(* CoDeSys 2.3.9.45 project: Stromsensor_01.pro *)
(* Libraries: SerComm.lib*31.5.11 08:54:36, Serial_Interface_01.lib*22.4.13 12:50:14, Modb_l05.lib*22.4.13 12:50:12, mod_com.lib*2.12.10 14:48:32, Standard.lib 20.5.14 08:13:26, Iecsfc.lib 16.5.13 14:00:50, SYSLIBCALLBACK.LIB 16.5.13 14:00:50 *)

(* Global variable list: Global_Constant *)
VAR_GLOBAL CONSTANT

	(*--- this values are possible parameters -> the real used quantity of sensors have to be smaller or equal ---*)
	MAX_SENSORS_PER_LINE		:	BYTE := 32;	(* max. quantity of possible slaves per line *)
	(*----------------------------------------------------------------------------------------------------------------------------------------------------------*)

END_VAR

(* Data type in line information/current sensor *)
TYPE typCurrentSensor :
	STRUCT
		rActualCurrent				:	REAL 	:= 0.0;	(* [A] actual  current *)
		rLimitErrorCurrent			:	REAL 	:= -3.0;	(* [A] threshold parameter for negative current error *)
		rInstalledCurrent			:	REAL 	:= 0.0; 	(* [A] installed nominal 125% current *)
		udErrorCounter			:	UDINT	:= 0;	(* error counter *)
		bErrorMaster				:	BYTE	:= 0;	(* communication error -> detected by the master *)
		bErrorSlave				:	BYTE	:= 0;	(* error at this sensor ->error generated and reprted by this slave *)

		bFillByte					:	BYTE 	:= 0;	(* fill byte to have an even byte count for this structure *)

		bSlaveAddress			:	BYTE	:= 0;	(* modbus address of this slave *)

		rBargraphValue			:	REAL 	:= 0.0;	(* value for Bargraph range -3.0 .. 80.0 *)


		xErrorMaster				:	BOOL;			(* error at this sensor -> see bErrorMaster *)
		xErrorSlave				:	BOOL;			(* error at this sensor -> see cErrorSlave *)
		xErrorOverflow				:	BOOL;			(* error at this sensor -> see 125% value *)
		xErrorUnderflow			:	BOOL;			(* error at this sensor -> see min. limit value *)
		xResetErrorCounter		:	BOOL;

		sDescription				:	STRING(25);	(* free userdefined description for this sensor *)
	END_STRUCT
END_TYPE

(* Data type in line information *)
TYPE typLineInfo :
	STRUCT
		Sensors 	:	ARRAY[1..MAX_SENSORS_PER_LINE] OF typCurrentSensor :=
									(*--- init values ------------------------------------------------------------------------------*)
									(rLimitErrorCurrent := -3.0, rInstalledCurrent := 29.8, bSlaveAddress := 1),
									(rLimitErrorCurrent := -3.0, rInstalledCurrent := 29.8, bSlaveAddress := 2),
									(rLimitErrorCurrent := -3.0, rInstalledCurrent := 29.8, bSlaveAddress := 3),
									(rLimitErrorCurrent := -3.0, rInstalledCurrent := 29.8, bSlaveAddress := 4),
									(rLimitErrorCurrent := -3.0, rInstalledCurrent := 29.8, bSlaveAddress := 5),
									(rLimitErrorCurrent := -3.0, rInstalledCurrent := 29.8, bSlaveAddress := 6),
									(rLimitErrorCurrent := -3.0, rInstalledCurrent := 29.8, bSlaveAddress := 7),
									(rLimitErrorCurrent := -3.0, rInstalledCurrent := 29.8, bSlaveAddress := 8),
									(rLimitErrorCurrent := -3.0, rInstalledCurrent := 29.8, bSlaveAddress := 9),
									(rLimitErrorCurrent := -3.0, rInstalledCurrent := 29.8, bSlaveAddress := 10),
									(rLimitErrorCurrent := -3.0, rInstalledCurrent := 29.8, bSlaveAddress := 11),
									(rLimitErrorCurrent := -3.0, rInstalledCurrent := 29.8, bSlaveAddress := 12),
									(rLimitErrorCurrent := -3.0, rInstalledCurrent := 29.8, bSlaveAddress := 13),
									(rLimitErrorCurrent := -3.0, rInstalledCurrent := 29.8, bSlaveAddress := 14),
									(rLimitErrorCurrent := -3.0, rInstalledCurrent := 29.8, bSlaveAddress := 15),
									(rLimitErrorCurrent := -3.0, rInstalledCurrent := 29.8, bSlaveAddress := 16),
									(rLimitErrorCurrent := -3.0, rInstalledCurrent := 29.8, bSlaveAddress := 17),
									(rLimitErrorCurrent := -3.0, rInstalledCurrent := 29.8, bSlaveAddress := 18),
									(rLimitErrorCurrent := -3.0, rInstalledCurrent := 29.8, bSlaveAddress := 19),
									(rLimitErrorCurrent := -3.0, rInstalledCurrent := 29.8, bSlaveAddress := 20),
									(rLimitErrorCurrent := -3.0, rInstalledCurrent := 29.8, bSlaveAddress := 21),
									(rLimitErrorCurrent := -3.0, rInstalledCurrent := 29.8, bSlaveAddress := 22),
									(rLimitErrorCurrent := -3.0, rInstalledCurrent := 29.8, bSlaveAddress := 23),
									(rLimitErrorCurrent := -3.0, rInstalledCurrent := 29.8, bSlaveAddress := 24),
									(rLimitErrorCurrent := -3.0, rInstalledCurrent := 29.8, bSlaveAddress := 25),
									(rLimitErrorCurrent := -3.0, rInstalledCurrent := 29.8, bSlaveAddress := 26),
									(rLimitErrorCurrent := -3.0, rInstalledCurrent := 29.8, bSlaveAddress := 27),
									(rLimitErrorCurrent := -3.0, rInstalledCurrent := 29.8, bSlaveAddress := 28),
									(rLimitErrorCurrent := -3.0, rInstalledCurrent := 29.8, bSlaveAddress := 29),
									(rLimitErrorCurrent := -3.0, rInstalledCurrent := 29.8, bSlaveAddress := 30),
									(rLimitErrorCurrent := -3.0, rInstalledCurrent := 29.8, bSlaveAddress := 31),
									(rLimitErrorCurrent := -3.0, rInstalledCurrent := 29.8, bSlaveAddress := 32);
									(*--------------------------------------------------------------------------------------------------*)
	END_STRUCT
END_TYPE

(* POU PLC_PRG, FBD *)
PROGRAM PLC_PRG
VAR RETAIN PERSISTENT
	SensorQuantity		:	BYTE := 1;			(* quantity of sensors -> 1 .. 32 *)
	Line					:	typLineInfo; 		(* table data *)
END_VAR
VAR
	mySensorLine		:	MODBUS_LINE;   (* communication fb *)
END_VAR
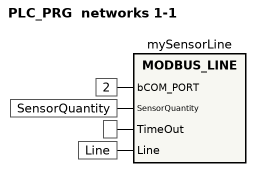
_FBD_ (* Function Block Diagram *)
NETWORK 1
	mySensorLine:MODBUS_LINE(bCOM_PORT: 2, SensorQuantity: SensorQuantity, TimeOut: , Line: Line)
_END_FBD_
END_PROGRAM

(* POU Line Communication/Single Line/MODBUS_LINE, ST *)
FUNCTION_BLOCK MODBUS_LINE
(*--- INTERFACE VARIABLES -------------------------------------------------------------------------------------*)
VAR_INPUT
	bCOM_PORT		:	BYTE := 2;
	SensorQuantity	:	BYTE := 1;			(* quantity of sensors *)
	TimeOut			:	TIME := t#30ms;	(* timeout for communication *)
END_VAR
VAR_IN_OUT
	Line				:	typLineInfo;		(**)
END_VAR
(*--- END INTERFACE VARIABLES ------------------------------------------------------------------------------*)

(*--- LOCAL VARIABLES --------------------------------------------------------------------------------------------*)
VAR
	MB_Master		:	MODBUS_MASTER_RTU;
	Query				:	typModbusQuery := (SlaveAddress := 1, FunctionCode := 3, StartAddress := 4, Quantity := 1, Data := 125(0) ); (* default values *)
	Start				:	BOOL;
	Response			:	typModbusResponse;

	JobNr				:	INT := 0;
	JobDelay			:	TON := (PT := t#30ms);
	i					:	INT;
	JobActive			:	BOOL;
END_VAR
(*--- delay between  two requests -----------------------*)
JobDelay(IN := NOT Start ); (*, PT := t#30ms);*)
(*-------------------------------------------------------------------*)

(*--- start a request  ------------------------------------------------------------------------------------*)
IF JobDelay.Q OR ((MB_Master.MB_Error = MB_TIME_OUT) AND NOT Start) THEN (* next job  *)
	JobNr := (JobNr MOD SensorQuantity) + 1;
	Query.SlaveAddress := Line.Sensors[JobNr].bSlaveAddress;

	Start := (Query.SlaveAddress <> 0);  (* if address <> 0 then start a request *)
	JobActive := Start;
END_IF
(*----------------------------------------------------------------------------------------------------------------------------*)

(*--- call the modbus master  ----------------------------------------------*)
MB_Master(	bCOM_PORT					:= bCOM_PORT,
				cbCOM_BAUDRATE			:= BAUD_19200,
				cpCOM_PARITY				:= PARITY_EVEN,
				csCOM_STOPBITS			:= STOPBITS_1,
				cbsCOM_BYTESIZE			:= BS_8,
				cfCOM_FLOW_CONTROL	:= HALFDUPLEX,
				TimeOut						:= TimeOut,
				StartFunction					:= Start,
				Query							:= Query,
				Response						:= Response);
(*------------------------------------------------------------------------------------*)

(*--- take over the response from sensor ----------------------------------------------------------------------------------------------*)
IF NOT Start AND (JobNr >= 1) AND (JobNr <= MAX_SENSORS_PER_LINE) AND JobActive THEN (* job is ready *)
	JobActive := FALSE;

	(*--- special process for  address 0 ------------------------------------------------------------*)
	IF Line.Sensors[JobNr].bSlaveAddress = 0  THEN (* Address = 0 -> erase errors *)
		Line.Sensors[JobNr].bErrorMaster 		:= 0;
		Line.Sensors[JobNr].bErrorSlave 		:= 0;
		Line.Sensors[JobNr].rActualCurrent 		:= 0.0; (* delete value  *)
		Line.Sensors[JobNr].rBargraphValue 	:= 0.0; (* delete bargraph *)
	(*----------------------------------------------------------------------------------------------------------*)

	ELSE (* take over the data  *)
		Line.Sensors[JobNr].bErrorMaster := INT_TO_BYTE(MB_Master.MB_Error);
		Line.Sensors[JobNr].bErrorSlave := WORD_TO_BYTE(Response.Error);

		IF MB_Master.MB_Error = MB_NO_ERROR THEN (* Job OK -> no errors -> take over the value  *)
			Line.Sensors[JobNr].rActualCurrent := INC_TO_AMPERE(Response.Data[0]); (* convert increments to ampere *)
			(*--- scale bargraph for 125%  -------------------------------------------------------------------------------------------------------------*)
			IF (Line.Sensors[JobNr].rInstalledCurrent > 0)  (* NO DIV 0 !!!  *)
			AND (Line.Sensors[JobNr].rActualCurrent > 0) THEN

				Line.Sensors[JobNr].rBargraphValue := (80.0 / Line.Sensors[JobNr].rInstalledCurrent) * Line.Sensors[JobNr].rActualCurrent;
			ELSE (* !! DIV durch NULL *)
				Line.Sensors[JobNr].rBargraphValue := Line.Sensors[JobNr].rActualCurrent;
			END_IF
			(*----------------------------------------------------------------------------------------------------------------------------------------------------*)

		ELSE (* error -> delete values *)
			Line.Sensors[JobNr].rActualCurrent 		:= 0.0;
			Line.Sensors[JobNr].rBargraphValue 	:= 0.0;

		END_IF
	END_IF

	ERROR_COUNTER; (* increment errorcounter  *)

END_IF

(*--- reset error counter ----------------------------------*)
FOR i := 1 TO SensorQuantity DO
	IF Line.Sensors[i].xResetErrorCounter THEN
		Line.Sensors[i].xResetErrorCounter := FALSE;
		Line.Sensors[i].udErrorCounter := 0;
	END_IF
END_FOR
(*---------------------------------------------------------------*)
END_FUNCTION_BLOCK
ACTION ERROR_COUNTER:
(*--- check for errors  --------------------------------------------------------------------------------------------------------------------------------------*)
Line.Sensors[JobNr].xErrorMaster 		:= (Line.Sensors[JobNr].bErrorMaster <> 0);
Line.Sensors[JobNr].xErrorSlave 		:= (Line.Sensors[JobNr].bErrorSlave <> 0);
Line.Sensors[JobNr].xErrorOverflow 		:= (Line.Sensors[JobNr].rActualCurrent > Line.Sensors[JobNr].rInstalledCurrent);
Line.Sensors[JobNr].xErrorUnderflow 	:= (Line.Sensors[JobNr].rActualCurrent < Line.Sensors[JobNr].rLimitErrorCurrent);

IF 	Line.Sensors[JobNr].xErrorMaster
	OR Line.Sensors[JobNr].xErrorSlave
	OR Line.Sensors[JobNr].xErrorOverflow
	OR Line.Sensors[JobNr].xErrorUnderflow
	 THEN (* increment error counter *)
	Line.Sensors[JobNr].udErrorCounter := Line.Sensors[JobNr].udErrorCounter + 1;
END_IF
END_ACTION

(* POU Line Communication/Single Line/Helper/INC_TO_AMPERE, ST *)
FUNCTION INC_TO_AMPERE : REAL
VAR_INPUT
	IN		:	WORD;
END_VAR
(* calculation from increments to ampere *)
INC_TO_AMPERE := (80.0 		(* max. current *)
                                       / 29126)	(* -> 32767 - 3641  Increments of the module for MAX_CURRENT *)
						* WORD_TO_INT(IN);
END_FUNCTION

(* Visualisation MASTER FOLIE/MASTERFOLIE
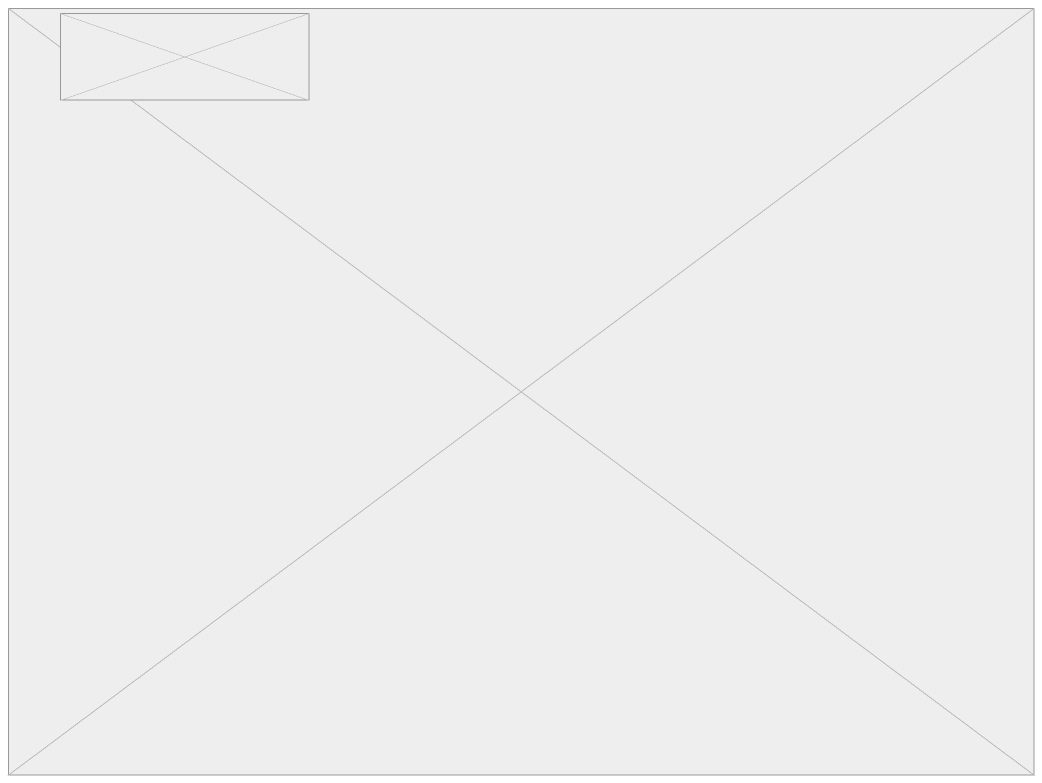
bitmap at (-1,0)-(1025,767): BILDER\789_620.BMP
bitmap at (51,5)-(300,92): BILDER\WAGO_INO.BMP
*)

(* Visualisation PLC_VISU
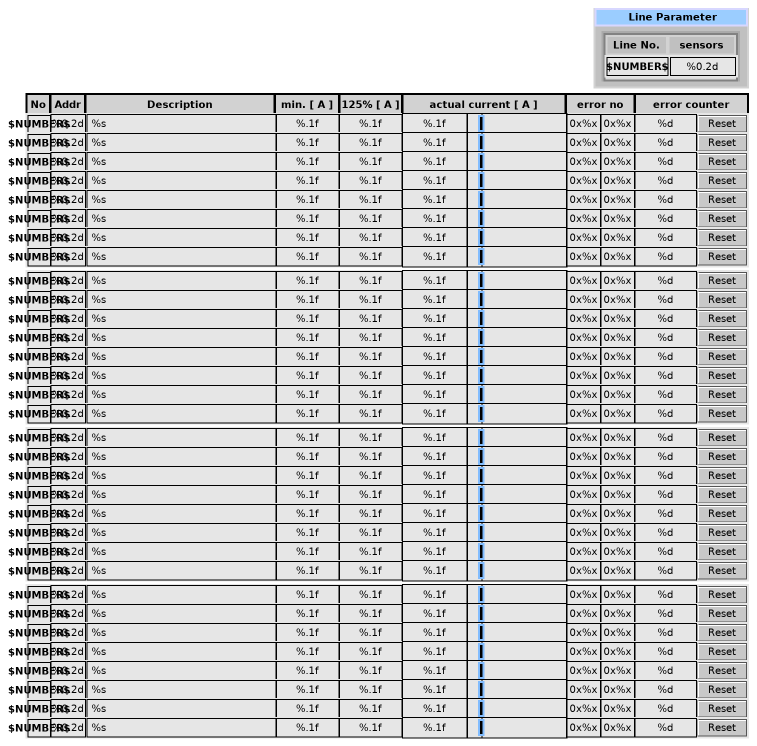
embedded screen at (51,92)-(774,116): VISU_TABLE_HEADLINE
embedded screen at (51,113)-(774,134): VISU_LINE
embedded screen at (51,132)-(774,153): VISU_LINE
embedded screen at (51,151)-(774,172): VISU_LINE
embedded screen at (51,170)-(774,191): VISU_LINE
embedded screen at (51,189)-(774,210): VISU_LINE
embedded screen at (51,208)-(774,229): VISU_LINE
embedded screen at (51,227)-(774,248): VISU_LINE
embedded screen at (51,246)-(774,267): VISU_LINE
embedded screen at (51,270)-(774,291): VISU_LINE
embedded screen at (51,289)-(774,310): VISU_LINE
embedded screen at (51,308)-(774,329): VISU_LINE
embedded screen at (51,327)-(774,348): VISU_LINE
embedded screen at (51,346)-(774,367): VISU_LINE
embedded screen at (51,365)-(774,386): VISU_LINE
embedded screen at (51,384)-(774,405): VISU_LINE
embedded screen at (51,403)-(774,424): VISU_LINE
embedded screen at (51,427)-(774,448): VISU_LINE
embedded screen at (51,446)-(774,467): VISU_LINE
embedded screen at (51,465)-(774,486): VISU_LINE
embedded screen at (51,484)-(774,505): VISU_LINE
embedded screen at (51,503)-(774,524): VISU_LINE
embedded screen at (51,522)-(774,543): VISU_LINE
embedded screen at (51,541)-(774,562): VISU_LINE
embedded screen at (51,560)-(774,581): VISU_LINE
embedded screen at (51,584)-(774,605): VISU_LINE
embedded screen at (51,603)-(774,624): VISU_LINE
embedded screen at (51,622)-(774,643): VISU_LINE
embedded screen at (51,641)-(774,662): VISU_LINE
embedded screen at (51,660)-(774,681): VISU_LINE
embedded screen at (51,679)-(774,700): VISU_LINE
embedded screen at (51,698)-(774,719): VISU_LINE
embedded screen at (51,717)-(774,738): VISU_LINE
group at (619,8)-(774,88)
  rectangle at (1,0)-(154,18): text "Line Parameter"
  rectangle at (12,27)-(74,47): text "Line No."
  rectangle at (74,27)-(142,47): text "sensors"
  embedded screen at (11,47)-(144,69): VISU_CONFIG_LINE
3 more shapes without text or variables
*)

(* Visualisation LINE/Elements/VISU_BARGRAPH
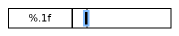
rectangle at (0,0)-(64,20): text "%.1f"; shows $CURRENT$
rectangle at (75,2)-(81,18): alarm colour if $CURRENT$ < 0; left $BARGRAPH_VALUE$; right $BARGRAPH_VALUE$
2 more shapes without text or variables
*)

(* Visualisation Elements/VISU_CONFIG_LINE
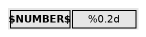
rectangle at (2,2)-(62,20): text "$NUMBER$"; tooltip Number of this sensor line
rectangle at (64,2)-(128,20): text "%0.2d"; shows $VALUE$; tooltip Quantity of used sensors at this line Range (1..32); editable 1..32
1 more shapes without text or variables
*)

(* Visualisation LINE/Elements/VISU_LINE
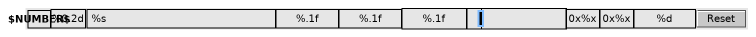
rectangle at (2,2)-(25,20): text "$NUMBER$"; tooltip line number
rectangle at (25,1)-(60,20): text "%0.2d"; shows $SENSOR$.bSlaveAddress; alarm colour if $SENSOR$.bSlaveAddress = 0; tooltip modbus address for this sensor range (1..32) if this address is equal zero then this line is not executed; editable 0..99
rectangle at (250,1)-(313,20): text "%.1f"; shows $SENSOR$.rLimitErrorCurrent; alarm colour if $SENSOR$.xErrorUnderflow; editable -10..+10
rectangle at (313,1)-(376,20): text "%.1f"; shows $SENSOR$.rInstalledCurrent; alarm colour if $SENSOR$.xErrorOverflow; editable 0..81
embedded screen at (376,0)-(541,21): VISU_BARGRAPH
rectangle at (540,1)-(574,20): text "0x%x"; shows $SENSOR$.bErrorMaster; alarm colour if $SENSOR$.xErrorMaster; tooltip error detected by the master ------------------------------------------------------------------ 16#00 -> no error 16#01 -> not supported function 16#90 -> extended slave error see slave 16#96 -> CRC error 16#97 -> illegal number of points 16#98 -> overrun response to long 16#99 -> time out no response from slave
rectangle at (608,1)-(670,20): text "%d"; shows $SENSOR$.udErrorCounter
button at (671,2)-(720,19): text "Reset"; toggles $SENSOR$.xResetErrorCounter; tooltip reset error counter
rectangle at (61,1)-(250,20): text "%s"; shows $SENSOR$.sDescription; tooltip free userdefined description max. length 25 characters; editable
rectangle at (574,1)-(608,20): text "0x%x"; shows $SENSOR$.bErrorSlave; alarm colour if $SENSOR$.xErrorSlave; tooltip error detected by the slave ------------------------------------------------------- 16#00 -> no error 16#65 -> underflow value < -10A 16#66 -> overflow value > +90A 16#67 -> invalid transfer function 16#68 -> invalid measuring
1 more shapes without text or variables
*)

(* Visualisation LINE/Elements/VISU_TABLE_HEADLINE
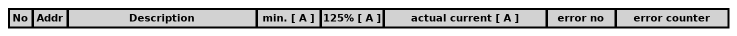
rectangle at (0,1)-(25,21): text "No"; tooltip line number
rectangle at (248,1)-(313,21): text "min. [ A ]"
rectangle at (312,1)-(376,21): text "125% [ A ]"
rectangle at (375,1)-(539,21): text "actual current [ A ]"
rectangle at (538,1)-(608,21): text "error no"
rectangle at (607,1)-(721,21): text "error counter"
rectangle at (24,1)-(60,21): text "Addr"; tooltip modbus address range (1..32)
rectangle at (59,1)-(249,21): text "Description"; tooltip free userdefined description max. length 25 characters
*)
